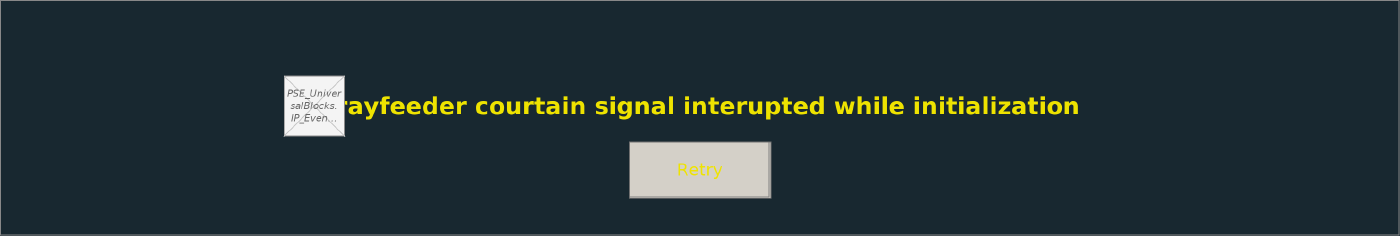
VISUALIZATION InitializingTrayfeederInterupted  // 1480x250
VAR_IN_OUT
	btnTrayfeederInitRetry : BOOL;
END_VAR
    Label (0,92 1480x40), "Trayfeeder courtain signal interupted while initialization"
    Image (300,80 64x64), image: PSE_UniversalBlocks.IP_EventSeverity.error
    Button (665,150 150x60), "Retry"
        toggle btnTrayfeederInitRetry
END_VISUALIZATION

(* stored: Version 1.1.0.1, ProductVersion 3.1.4024.9
   Visu InitializingTrayfeederInterupted: Id {1f6eb996-122d-47fe-b7dd-036f8b701875} *)
